ABB RobotStudio station: stazione_base_20221027-105558.rsstn

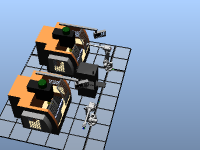
Station Station (saved by RobotStudio 7.0.8504.151)
Controller Controller7, task T_ROB2: task frame (RAPID world) sits at (2603.59, 0, 0) mm in the station
Controller Controller7, task T_ROB1: task frame (RAPID world) sits at (2603.59, 0, 0) mm in the station
Controller Controller7
  mechanical unit ROB_1: IRB4600_20_250_C_01, 6 joints, base frame (-2603.59, 0, 0) mm
  mechanical unit ROB_2: IRB4600_20_250_C_01_2, 6 joints, base frame (1396.41, 0, 0) mm
Layout (positions relative to the parent item):
  - IRB4600_20_250_C_01 [mechanism, from Robots\IRB4600_20_250_C_G_01.rslib] at (0, 0, 0) mm; joint values [-1.5269, -0.0965, 0.041, 0.0078, 1.4594, -3.138] (rad or m)
  - IRB4600_20_250_C_01_2 [mechanism, from Robots\IRB4600_20_250_C_G_01.rslib] at (4000, 0, 0) mm; joint values [0, 0, 0, 0, 0.5236, 0] (rad or m)
  - CNC [part] at (0, -3500, 0) mm, rotated rx 90 ry 0 rz 0 deg
  - CNC_2 [part] at (4000, -3500, 0) mm, rotated rx 90 ry 0 rz 0 deg
  - Macchina_Test [part] at (0, -1000, 860) mm, rotated rx 90 ry 0 rz 90 deg
